PROGRAM OP120_JB_IO
VAR
OP120_JB_DI_MODULE_1 AT %I* : WORD;
OP120_JB_DI_MODULE_2 AT %I* : WORD;

OP120_JB_DO_MODULE_1 AT %Q* : WORD;
OP120_JB_DO_MODULE_2 AT %Q* : WORD;

	WORD_AS_BIT_0: WORD_AS_BIT;
	WORD_AS_BIT_1: WORD_AS_BIT;
	
	BIT_AS_WORD_0: BIT_AS_WORD;
	BIT_AS_WORD_1: BIT_AS_WORD;
END_VAR

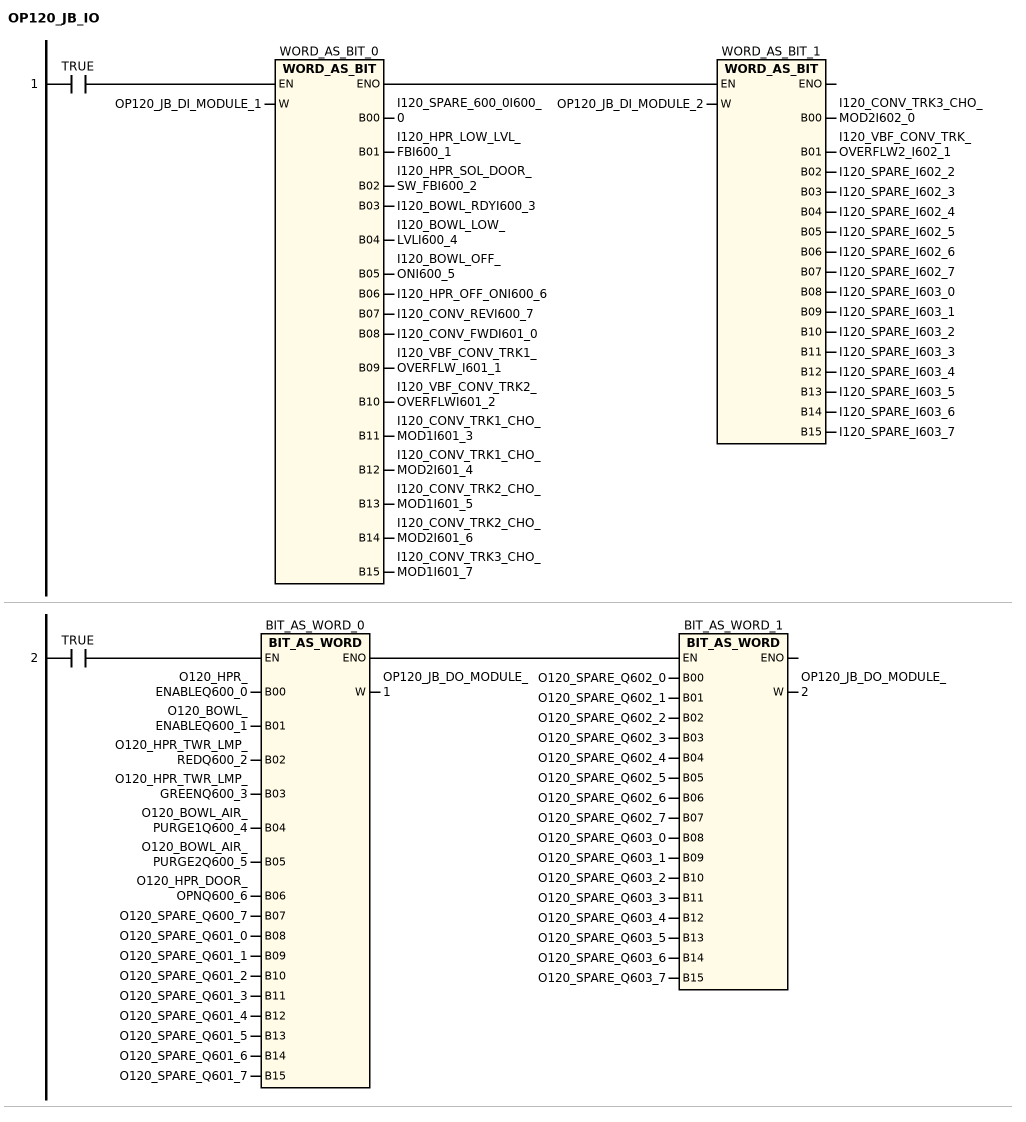
// NETWORK 1
WORD_AS_BIT_0(
    W := OP120_JB_DI_MODULE_1,
    B00 => I120_SPARE_600_0I600_0,
    B01 => I120_HPR_LOW_LVL_FBI600_1,
    B02 => I120_HPR_SOL_DOOR_SW_FBI600_2,
    B03 => I120_BOWL_RDYI600_3,
    B04 => I120_BOWL_LOW_LVLI600_4,
    B05 => I120_BOWL_OFF_ONI600_5,
    B06 => I120_HPR_OFF_ONI600_6,
    B07 => I120_CONV_REVI600_7,
    B08 => I120_CONV_FWDI601_0,
    B09 => I120_VBF_CONV_TRK1_OVERFLW_I601_1,
    B10 => I120_VBF_CONV_TRK2_OVERFLWI601_2,
    B11 => I120_CONV_TRK1_CHO_MOD1I601_3,
    B12 => I120_CONV_TRK1_CHO_MOD2I601_4,
    B13 => I120_CONV_TRK2_CHO_MOD1I601_5,
    B14 => I120_CONV_TRK2_CHO_MOD2I601_6,
    B15 => I120_CONV_TRK3_CHO_MOD1I601_7); // WORD_AS_BIT
WORD_AS_BIT_1(
    W := OP120_JB_DI_MODULE_2,
    B00 => I120_CONV_TRK3_CHO_MOD2I602_0,
    B01 => I120_VBF_CONV_TRK_OVERFLW2_I602_1,
    B02 => I120_SPARE_I602_2,
    B03 => I120_SPARE_I602_3,
    B04 => I120_SPARE_I602_4,
    B05 => I120_SPARE_I602_5,
    B06 => I120_SPARE_I602_6,
    B07 => I120_SPARE_I602_7,
    B08 => I120_SPARE_I603_0,
    B09 => I120_SPARE_I603_1,
    B10 => I120_SPARE_I603_2,
    B11 => I120_SPARE_I603_3,
    B12 => I120_SPARE_I603_4,
    B13 => I120_SPARE_I603_5,
    B14 => I120_SPARE_I603_6,
    B15 => I120_SPARE_I603_7); // WORD_AS_BIT

// NETWORK 2
BIT_AS_WORD_0(
    B00 := O120_HPR_ENABLEQ600_0,
    B01 := O120_BOWL_ENABLEQ600_1,
    B02 := O120_HPR_TWR_LMP_REDQ600_2,
    B03 := O120_HPR_TWR_LMP_GREENQ600_3,
    B04 := O120_BOWL_AIR_PURGE1Q600_4,
    B05 := O120_BOWL_AIR_PURGE2Q600_5,
    B06 := O120_HPR_DOOR_OPNQ600_6,
    B07 := O120_SPARE_Q600_7,
    B08 := O120_SPARE_Q601_0,
    B09 := O120_SPARE_Q601_1,
    B10 := O120_SPARE_Q601_2,
    B11 := O120_SPARE_Q601_3,
    B12 := O120_SPARE_Q601_4,
    B13 := O120_SPARE_Q601_5,
    B14 := O120_SPARE_Q601_6,
    B15 := O120_SPARE_Q601_7,
    W => OP120_JB_DO_MODULE_1); // BIT_AS_WORD
BIT_AS_WORD_1(
    B00 := O120_SPARE_Q602_0,
    B01 := O120_SPARE_Q602_1,
    B02 := O120_SPARE_Q602_2,
    B03 := O120_SPARE_Q602_3,
    B04 := O120_SPARE_Q602_4,
    B05 := O120_SPARE_Q602_5,
    B06 := O120_SPARE_Q602_6,
    B07 := O120_SPARE_Q602_7,
    B08 := O120_SPARE_Q603_0,
    B09 := O120_SPARE_Q603_1,
    B10 := O120_SPARE_Q603_2,
    B11 := O120_SPARE_Q603_3,
    B12 := O120_SPARE_Q603_4,
    B13 := O120_SPARE_Q603_5,
    B14 := O120_SPARE_Q603_6,
    B15 := O120_SPARE_Q603_7,
    W => OP120_JB_DO_MODULE_2); // BIT_AS_WORD

END_PROGRAM

(* stored: Version 1.1.0.1, ProductVersion 3.1.4024.11
   POU OP120_JB_IO: Id {f7c0b7bb-5cf9-4367-adad-b8fd389c56b3}, SpecialFunc None *)
